TYPE ST_Ampel_Parameter :
STRUCT
	AutoQuittierung			: BOOL;
END_STRUCT
END_TYPE

(* stored: Version 1.1.0.1, ProductVersion 3.1.4024.9
   DUT ST_Ampel_Parameter: Id {ee7f39ae-6119-4e06-aeb9-f8dbdfdfa1ec} *)
